// TIA Portal V20 export
TYPE "HMI_OpAnL"
   STRUCT
      SP_ExtOp : Bool := FALSE;   // Operator input to select external setpoint
      SP_IntOp : Bool := TRUE;   // Operator input to select internal setpoint
      SP_Int : Real := 0.0;   // Internal Analog setpoint
      SP_Ext : Real;   // External Analog setpoint
      SP_HiLim : Real := 100.0;   // Input High Limit
      SP_LoLim : Real := 0.0;   // Input Low Limit
      SP_OpScale : "ScaVal";   // SP- Bar Display Limits for OS
      SP_Unit : Int := 1001;   // Engineering units of Input
      PV_In : Real;   // Feedback Analog Input
      PV_In_ST : Byte := BYTE#16#80;   // PV_In Signal Status
      PV_OpScale : "ScaVal";   // PV- Bar Display Limits for OS
      PV_Unit : Int := 1001;   // Engineering units of Feedback Input
      SP_TrkExt : Bool := FALSE;   // 1: SP_Int tracks SP_Ext in External
      SP_UpRaLim : Real := 100.0;   // Upward rate limit for setpoint
      SP_DnRaLim : Real := 100.0;   // Downward rate limit for setpoint
      SP_RateOn : Bool := FALSE;   // 1= Activate limitation of setpoint gradients
      SP_RmpOn : Bool := FALSE;   // 1= Activate setpoint ramp to target SP_RmpTarget
      SP_RmpModTime : Bool := FALSE;   // 1= Use time SP_RmpTime for ramp, 0= Use rates SP_UpRaLim, SP_DnRaLim
      SP_RmpTime : Real := 0.0;   // Setpoint ramp time [s,min,h]
      SP_RmpTarget : Real := 0.0;   // Setpoint ramp target
      OnOp : Bool := FALSE;   // 1=On Mode: On Mode by Operator
      OosOp : Bool := FALSE;   // 1=Oos Mode: Oos Mode by Operator
      TimeFactor : Int := 0;   // Time Conversion Factor (0- Sec, 1- Min, 2- Hour)
      BatchID : DWord := 16#0;   // Current Batch ID (number)
      BatchName : String[32] := '';   // Current Batch Name
      StepNo : DWord := 16#0;   // Batch Step Number
      SP_Out { ExternalWritable := 'False'} : Real;   // Analog Output Value
      SP_RateTarget { ExternalWritable := 'False'} : Real := 0.0;   // Target for limitation of setpoint gradients
      SP_RemRT { ExternalWritable := 'False'} : Real := 0.0;   // Remaining ramp time of setpoint
      OS_PermOut { ExternalWritable := 'False'} : DWord := DWORD#16#FFFF_FFFF;   // Operator Permission: Output for OS
      OS_PermLog { ExternalWritable := 'False'} : DWord := DWORD#16#FFFF_FFFF;   // Operator Permission: Output for OS
      OpSt_Out { ExternalWritable := 'False'} : DWord := 16#0;   // Enabled operator stations
      ST_Worst { ExternalWritable := 'False'} : Byte := 16#80;   // Worst Signal Status
      Status1 { ExternalWritable := 'False'} : DWord := 16#0;   // Status Word1
      AlarmState { ExternalWritable := 'False'} : Word;   // Alarm State for group display / Alarm Status for group display
   END_STRUCT;
   // // SP_OpScale.High : High Value
   // // SP_OpScale.Low : Low Value
   // // PV_OpScale.High : High Value
   // // PV_OpScale.Low : Low Value
END_TYPE
